// SIMATIC S7-200 SMART project (STEP 7-Micro/WIN SMART), CPU SR40

SYMBOL_TABLE 系统符号
First_Scan_On    SM0.1    // 仅在第一个扫描周期时接通
Clock_1s         SM0.5    // 针对 1 s 的周期时间，时钟脉冲接通 0.5 s，断开 0.5 s.
END_SYMBOL_TABLE

ORGANIZATION_BLOCK MAIN:OB1
TITLE=程序注释
BEGIN
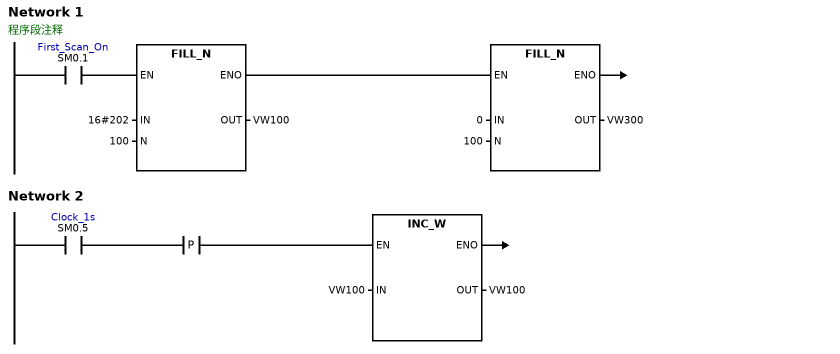
Network 1
// 程序段注释
// (network saved uncompiled; LAD cells follow)
// row 0: c0 -| |- First_Scan_On:SM0.1  c1 [FILL_N EN:=power@row0, IN:=16#202, N:=100, ENO=>power, OUT=>VW100]  c2 --  c3 --  c4 [FILL_N EN:=power@row0, IN:=0, N:=100, ENO=>power, OUT=>VW300]  c5 ->
// row 1: c1 [box]  c4 [box]
Network 2
LD     Clock_1s:SM0.5
EU
INCW   VW100
Network 3
// 程序段注释
END_ORGANIZATION_BLOCK
